TYPE TcoInsightSoftEventControl_v_5_x_x :
STRUCT
	TriggerSoftEventAcknowledge AT %I* : ARRAY [0..7] OF BOOL;
	TriggerSoftEvent AT %Q* : ARRAY [0..7] OF BOOL;	
END_STRUCT
END_TYPE

(* stored: Version 1.1.0.1, ProductVersion 3.1.4024.11
   DUT TcoInsightSoftEventControl_v_5_x_x: Id {7792c4e9-0f72-01e8-0d88-da5811ee8506} *)
